// Contains string constants for working with files
{attribute 'no_explicit_call' := 'Body contains no logic, calling methods only allowed.'}
{attribute 'hide_all_locals'}
PROGRAM Constants
VAR
	_pathSeperators	: FB_PathSeperators;	
	_wildcards	: FB_Wildcards;
END_VAR

// Returns WINDOWS path separator "/"
PROPERTY PathSeperators : REFERENCE TO FB_PathSeperators
GET
PathSeperators REF= _pathSeperators;
END_GET
END_PROPERTY

PROPERTY Wildcards : REFERENCE TO FB_Wildcards
GET
Wildcards REF= _wildcards;
END_GET
END_PROPERTY

END_PROGRAM

(* stored: Version 1.1.0.1, ProductVersion 3.1.4024.14
   POU Constants: Id {ff96902c-5136-0ae0-1075-e89641639929}, SpecialFunc None
   Property PathSeperators: Id {79e1fca6-79e7-07e8-052c-4d9c7cd66fd4}
   Get Get: Id {e5c4fede-1050-0288-3d07-af087dead439}
   Property Wildcards: Id {205ac2e7-93f7-0748-2d16-c4c53b0f5d9e}
   Get Get: Id {1e9a9c22-2a62-021e-0029-6d9c07909dea} *)
